// TIA Portal project "Lab2-S7" (V15.1)

(* hardware
DEVICE "S7-1200 station_1"  S7-1200 Station
   slot 0: "Rack_0"  S7-1200 Rack  Rack  V1.0
   slot 1: "PLC_1"  CPU 1214C AC/DC/Rly  6ES7 214-1BG40-0XB0  V4.2
*)

// ===== PLC "PLC_1"  CPU 1214C AC/DC/Rly =====

VAR_GLOBAL   // PLC tag table "Tabla de variables estándar"
   "Clock_Byte" AT %MB0 : Byte;
   "Clock_10Hz" AT %M0.0 : Bool;
   "Clock_5Hz" AT %M0.1 : Bool;
   "Clock_2.5Hz" AT %M0.2 : Bool;
   "Clock_2Hz" AT %M0.3 : Bool;
   "Clock_1.25Hz" AT %M0.4 : Bool;
   "Clock_1Hz" AT %M0.5 : Bool;
   "Clock_0.625Hz" AT %M0.6 : Bool;
   "Clock_0.5Hz" AT %M0.7 : Bool;
   "System_Byte" AT %MB1 : Byte;
   "FirstScan" AT %M1.0 : Bool;
   "DiagStatusUpdate" AT %M1.1 : Bool;
   "AlwaysTRUE" AT %M1.2 : Bool;
   "AlwaysFALSE" AT %M1.3 : Bool;
   "Tag_1" AT %I0.0 : Bool;
   "Tag_2" AT %M2.0 : Bool;
   "Tag_3" AT %M2.1 : Bool;
END_VAR

DATA_BLOCK "LOGO_S7"   // DB1
{ S7_Optimized_Access := 'FALSE' }
VERSION : 0.1
   VAR
      I1 : Bool;
      I2 : Bool;
      I3 : Bool;
      I4 : Bool;
      I5 : Bool;
      I6 : Bool;
      I7 : Bool;
      I8 : Bool;
      Q1 : Bool;
      Q2 : Bool;
      Q3 : Bool;
      Q4 : Bool;
      VW2 : Int;
      VW4 : Int;
   END_VAR
BEGIN
END_DATA_BLOCK

FUNCTION "FC_LOGO_S7" : Void   // FC1, FBD
{ S7_Optimized_Access := 'TRUE' }
VERSION : 0.1
   VAR_TEMP   // added for the SCL form of the ladder/FBD networks
      _w1 : Bool;
   END_VAR
BEGIN

REGION Network 1: Activar salida Q1 del Logo8 desde la entrada I0.0 o la Marca 2.0 del PLC S7-1200
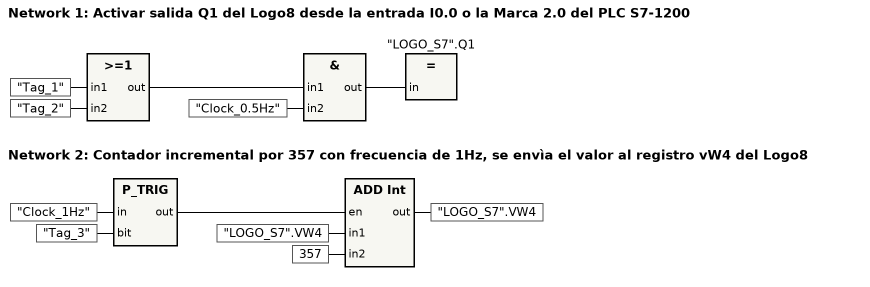
   "LOGO_S7".Q1 := ("Tag_1" OR "Tag_2") AND "Clock_0.5Hz";
END_REGION

REGION Network 2: Contador incremental por 357 con frecuencia de 1Hz, se envìa el valor al registro vW4 del Logo8
   #_w1 := "Clock_1Hz" AND NOT "Tag_3";   // rising edge
   "Tag_3" := "Clock_1Hz";
   IF #_w1 THEN "LOGO_S7".VW4 := "LOGO_S7".VW4 + 357; END_IF;
END_REGION
END_FUNCTION

ORGANIZATION_BLOCK "Main"   // OB1, LAD, ProgramCycle
TITLE = "Main Program Sweep (Cycle)"
{ S7_Optimized_Access := 'TRUE' }
VERSION : 0.1
   VAR_INPUT
      Initial_Call : Bool;   // Initial call of this OB
      Remanence : Bool;   // =True, if remanent data are available
   END_VAR
BEGIN

REGION Network 1
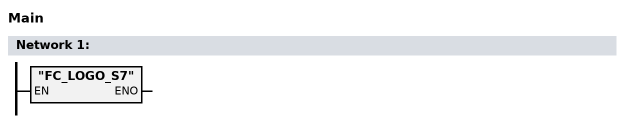
   RUNG wire#powerrail
      "FC_LOGO_S7"()
   END_RUNG
   // the same network as SCL:
   "FC_LOGO_S7"();
END_REGION
END_ORGANIZATION_BLOCK